(* Logix 5000 project; controller BWFG_Project vendor 1 type 14 code 92 rev 20.13; software revision 20.04 *)

TASK MainTask (continuous, watchdog 500 ms) : MainProgram

MODULES
   Local : vendor 1 type 14 code 92 (ICP 5, rev 20.13)
      DNET_Scanner : vendor 1 type 12 code 14 (ICP 11, rev 7.3, Output RPI 20 ms, Input RPI 20 ms)
      Servo_Module : 1756-M02AE (ICP 12, rev 20.2, MotionAsync RPI 25 ms, MotionEvent RPI 1000 ms, MotionSync RPI 2 ms)
      Ethenet_Module : 1756-EN2T (Ethernet 10.100.88.20, ICP 9, rev 10.7)   // CLX Etherent Module
         PF70 : vendor 1 type 123 code 48 (Ethernet 10.100.88.53, rev 2.9, Output RPI 20 ms)
              PF70:O.DRIVELOGICRSLT_START   // ENET Speed Start
              PF70:O.DRIVELOGICRSLT_REVERSE   // ENET Rev Start
              PF70:O.DRIVELOGICRSLT_FORWARD   // Enet FWD Start
             : vendor 1 type 123 code 8192 (DPI 5, rev 5.2)
      DHRIO : 1756-DHRIO (ICP 10, rev 5.4, Input RPI 25 ms)
         Flex_Rack : 1794-ASB (RIO 0, rev 1.1, Output RPI 16 ms)   // Flex RIO Rack in Workcell
         Robot_Rack : 1794-ASB (RIO 8, rev 1.1, Output RPI 48 ms)
END_MODULES

VAR_GLOBAL   (* controller tags *)
   Amber_Stack_LT : ALIAS FOR Flex_Rack:O.Data[3].1;   // The Amber stack Light
   Auto_mode : BOOL;   // Auto Mode Trigger ON/OFF
   Axis_0 : AXIS_SERVO;
   B3 : DINT;   // Hold value for robot Info
        .4   // Lift Locate Lower Cycle (AUTO)
        .0   // Permit Auto Mode
        .3   // Pallet Discarge Cycle
        .5   // Lift locate lower cycle auto
   Barcode_char : SINT[12] := ([0] := 110, [1] := 114, [2] := 32, [3] := 32, [4] := 32, [5] := 32, [6] := 32, [7] := 32, [8] := 32, [9] := 32, [10] := 32, [11] := 32);   // Barcode scanned info
   Barcode_Delay : BOOL;   // Delay created for barcode to allow info to be scanned then sent
   Barcode_Display : SINT[12] := ([0] := 62, [1] := 66, [2] := -16, [3] := -16, [4] := -16, [5] := -16, [6] := -16, [7] := -16, [8] := -16, [9] := -16, [10] := -16, [11] := -16);   // display the barcode value after info been translated from Asscii to decimal
   Barcode_OneShot : BOOL;   // a Oneshot for barcode to be sent
   Barcode_PB : BOOL;   // Push Button to Trigger the Barcode For manual mode and testing
   Barcode_Raw : STRING;   // Barcode Raw data (in ASCII)
   Barcode_Read_Done : BOOL := 1;   // Barcode signal it's done scanning
   Binary : DINT;
   Bottle_Control : CONTROL := (LEN := 5, EM := 1);   // Control for Bottle FiFo
   Bottle_FIFO : SINT[5];   // Bottle Fifo to Hold and send the list of Bottle value info (diffrent types of 12)
   BottleType : INT;   // Type of Bottle Given to be drawned
   Cabernet_Total : REAL := 100.0;
   Cell_Power_ON : ALIAS FOR Flex_Rack:I.Data[0].0;   // Workcell Power On Input
   Cell_Stop_PB : ALIAS FOR Flex_Rack:I.Data[1].11;   // Workcell Stop PB
   Champagne_Total : REAL := 100.0;
   Clear_Out_Oneshot : BOOL;   // Clear the Outputs when switching manual entry modes
   Cycle_Complete : ALIAS FOR Robot_Rack:I.Data[0].2;   // Cycle Complete Signal
   Cycle_Start : ALIAS FOR Robot_Rack:O.Data[0].0;   // Cycle start Trigger
   Direction_Mask_Value : DINT := 47;   // the Diresctional Mask for the VFD to change it From Ethernet to Deffalt
   Display_N : DINT[12];
   Display_PV : DINT;   // the Display PV screen, used to change the screen
   DNET_MODE_Select : BOOL;
   Drive_Actual_FWD_Speed : REAL;   // Real Speed of the FWD of the driver (in HZ)
   Drive_Actual_REV_Speed : REAL;   // Real Speed of the REV of the driver (in HZ)
   Drive_REQ_SPD_A : REAL;   // Driver running Indicator
   Drive_Running_IND : BOOL;   // the speed request for the driver in HZ
   Drive_SPD_Request : REAL;
   ENET_FWD_Speed : DINT;   // the set fwd speed
   ENET_REV_Speed : DINT;   // The set REV speed
   Enet_speed_convert : DINT;
   Enet_Speed_HOLD : DINT;
   Ent_Stop_Bit : ALIAS FOR Flex_Rack:O.Data[3].5;   // Ethernet Stop BIT
   Entrance_Convr_Message : SINT := 1;   // PV1000+ Entrance Conveyor Message 1=Stopped, 2=Forward 3=Reverse
   Entrance_FWD_PB : BOOL;   // PV1000+ ENTRANCED CONVEYOR FORWARD PB MANUAL SCREEN
   Entrance_REV_PB : BOOL;   // PV1000+ ENTRANCED CONVEYOR REVERSE PB MANUAL SCREEN
   Entrance_Speed_FPM : REAL;   // PV1000+ ENTRANCE CONVEYOR SPEED FEET-PER-MIN
   Entrance_Speed_Select : SINT := 5;
        .0   // PV1000+ Entrance Conveyor VFD Speed Select Bit 0
        .1   // PV1000+ Entrance Conveyor VFD Speed Select Bit 1
        .2   // PV1000+ Entrance Conveyor VFD Speed Select Bit 2
   Entrance_Speed_Timer : TIMER := (PRE := 5000);   // 5 second timer (1/12 of a minute)
        .DN   // 5 second timer (1/12 of a minute)
   Entrance_Sprocket_Pulse_Prox : ALIAS FOR Flex_Rack:I.Data[0].13;   // ENTRANCE CONVEYOR SPROCKET PULSE PROX 1 PULSE = 0.842 INCHES
   Event_Driven_Timer : TIMER[14] := ([0].PRE := 500, [1].PRE := 500, [2].PRE := 1700, [3].PRE := 500, [4].PRE := 500, [5].PRE := 500, [6].PRE := 500, [7].PRE := 500, [8].PRE := 500, [9].PRE := 500, [10].PRE := 500, [11].PRE := 500, [12].PRE := 500, [13].PRE := 2000);
   fault_servo_Reset : BOOL;
   FIFO_Bottle_Input : SINT := -16;
   FIFO_Bottle_Output : SINT := 1;
   FIFO_Level_Input : SINT := 96;
   FIFO_Level_Output : SINT := 55;
   FIFO_Location_Input : SINT := 66;
   FIFO_Location_Output : SINT := 1;
   FIFO_Wine_Input : SINT := -16;
   FIFO_Wine_Output : SINT := 1;
   Fill_Hold_percent : REAL := -160.0;   // holds percent values to then be sent as a whole value
   Fill_Level : INT;
   Fully_stop : BOOL;   // E_Stop LT
   FWD_REV_Mode : BOOL := 1;   // 0=FWD 1= REV
   Gate_Convr_FWD_PB : BOOL;   // PV1000+ GATE CONVEYOR FORWARD PB MANUAL SCREEN
   Gate_Convr_Message : SINT := 1;   // PV1000+ Gate Conveyor Message Display 1=Stopped 2=Forward 3=Reverse
   Gate_Convr_REV_PB : BOOL;   // PV1000+ GATE CONVEYOR REVERSE PB MANUAL SCREEN
   Gate_FS : BOOL;
   Gate_FWD_Starter : ALIAS FOR Flex_Rack:O.Data[4].2;   // Gate Conveyor Forward Motor Starter
   Gate_FWD_Starter_Contact : ALIAS FOR Flex_Rack:I.Data[1].5;   // Gate Conveyor Auxilary Contact Motor Forward Starter
   Gate_PL : ALIAS FOR Flex_Rack:O.Data[4].4;
   Gate_REV_Starter : ALIAS FOR Flex_Rack:O.Data[4].3;   // Gate Conveyor Reverse Motor Starter
   Gate_REV_Starter_Contact : ALIAS FOR Flex_Rack:I.Data[1].6;   // Gate Conveyor Auxilary Contact Motor Reverse Starter
   Gate_RS : BOOL;
   GIN : ALIAS FOR Robot_Rack:O.Data[0];
   Go_to_Auto_PB : BOOL;   // PV1000+ AUTO SCREEN SELECTED
   GO_to_Display_PB : BOOL;   // PV1000+ DISPALY SCREEN SELECTED
   Go_to_Robot : BOOL;   // PV1000+ ROBOT SCREEN SELECTED
   Go_To_Speed : BOOL;
   Go_to_Tracking : BOOL;   // PV1000+ TRACKING SCREEN SELECTED
   Goto_Main_PB : BOOL;   // PV1000+ MAIN SCREEN SELECTED
   Goto_Manual_PB : BOOL;   // PV1000+ MANUAL SCREEN SELECTED
   Green_Stack_LT : ALIAS FOR Flex_Rack:O.Data[3].2;
   HMI_indexer : SINT;
   Home_PB : BOOL;
   In_Cycle : ALIAS FOR Robot_Rack:I.Data[0].1;
   Input_clear_oneshot : BOOL;
   Level_Control : CONTROL := (LEN := 5, EM := 1);
   Level_FIFO : SINT[5];
   Level_Percent : REAL := 5.5;
   Lift_Locate_DOWN_Prox : ALIAS FOR Flex_Rack:I.Data[1].3;   // Lift Locate Down Prox
   Lift_Locate_Lower_Prox : ALIAS FOR Flex_Rack:I.Data[1].3;
   Lift_Locate_Message : SINT := 1;   // PV1000+ Lift-Locate-Unit Message Display 1=Lowered, 2=Raised
   Lift_Locate_PB : BOOL;   // PV1000+ Lift Locate PB (maintained)
   Lift_Locate_Prox : ALIAS FOR Flex_Rack:I.Data[1].1;
   Lift_Locate_Raised_Prox : ALIAS FOR Flex_Rack:I.Data[1].2;
   Lift_Locate_UP_Prox : ALIAS FOR Flex_Rack:I.Data[1].2;   // Lift Locate UP Prox
   Lift_Lower_Solenoid : ALIAS FOR Flex_Rack:O.Data[4].1;   // Lift Locate Lower Solenoid
   Lift_Raise_Solenoid : ALIAS FOR Flex_Rack:O.Data[4].0;   // Lift Locate Raise Solenoid
   Load_PB : BOOL;
   Location : INT;
   Location_Control : CONTROL := (LEN := 5, EM := 1);
   Location_FIFO : SINT[5];
   LTU_B : BOOL;
   LTU_DOWN_Prox : ALIAS FOR Flex_Rack:I.Data[0].10;   // Lift-transfer-Unit Down Prox
   LTU_Lower_Prox : ALIAS FOR Flex_Rack:I.Data[0].10;
   LTU_Lower_Solenoid : ALIAS FOR Flex_Rack:O.Data[3].12;   // Lift-Transfer-Unit Lower Solenoid
   LTU_Message : SINT := 2;   // PV1000+ Lift-Transfer-Unit Message Display 1=Lowered, 2=Centre 3=Raised
   LTU_Mid : BOOL;
   LTU_Posn_Select : SINT := 2;
        .0   // PV1000+ LTU Position Selector Bit 0
        .1   // PV1000+ LTU Position Selector Bit 1
   LTU_Prox : ALIAS FOR Flex_Rack:I.Data[0].9;
   LTU_Raise_Solenoid : ALIAS FOR Flex_Rack:O.Data[3].11;   // Lift-Transfer-Unit Raise Solenoid
   LTU_Raised_Prox : ALIAS FOR Flex_Rack:I.Data[0].11;
   LTU_Top : BOOL;
   LTU_UP_Prox : ALIAS FOR Flex_Rack:I.Data[0].11;   // Lift-transfer-Unit UP Prox
   Main_Screen_Button : BOOL;   // PV1000+ MAIN SCREEN SELECTED
   Man_Barcode_ON : BOOL;   // Allows the barcode to be turn on when running in manual mode for testing
   Man_Bottle : DINT := 1;
   Man_Level : DINT := 55;
   Man_Load_PB : BOOL;   // Loads the manual enetry values
   Man_Location : DINT := 1;
   Man_Mode : BOOL;
   Man_Mode_ON : BOOL;   // PV1000+ MANUAL MODE INDICATOR
   Man_Wine : DINT := 1;
   Manual_Enty : BOOL := 1;   // allows manual entry for orders
   manual_Screen_button : BOOL;   // PV1000+ Manual SCREEN SELECTED
   Merlot_Total : REAL := 94.5;
   Motion_Group_One : MOTION_GROUP;
   MSG_Display_Num : COUNTER := (PRE := 300, ACC := 154);
   MSG_Timer : TIMER := (PRE := 50, ACC := 41, EN := 1, TT := 1);
   MSG_Timer_2 : TIMER := (PRE := 50, EN := 1, TT := 1);
   New_Message_Sent_N : ALIAS FOR Local:11:I.Data[0].15;
   One_Shot : BOOL;
   One_Shot_Mid : BOOL;
   One_Shot_Rise : BOOL;
   OneShot_Clear_bits : BOOL;
   pallet_at_gate : ALIAS FOR Flex_Rack:I.Data[2].4;
   PF70_Fault_Reset : BOOL;
   PF70_Feedback_Speed_FWD_Hz : REAL;
   PF70_Feedback_Speed_REV_Hz : REAL;
   PF70_Parameter_Value : INT[300] := ([2] := 400, [10] := 2358, [12] := 8337, [13] := 8339, [16] := -6, [17] := 57, [26] := 37, [27] := 6000, [28] := 9, [29] := 2009, [41] := 5750, [42] := 5, [43] := 600, [44] := 1700, [45] := 21, [46] := 1, [47] := 300, [48] := 356, [54] := 5750, [55] := 1300, [56] := 3, [61] := 3, [62] := 237, [63] := 25, [69] := 219, [70] := 219, [71] := 1150, [72] := 150, [82] := 700, [83] := 100, [90] := 1, [91] := 700, [93] := 22, [94] := 700, [96] := 1, [97] := 600, [100] := 100, [101] := 50, [102] := 100, [103] := 200, [104] := 300, [105] := 400, [106] := 500, [107] := 600, [117] := 2, [119] := 600, [121] := 1000, [122] := 400, [127] := 5000, [128] := 4866, [129] := 200, [130] := 100, [131] := -1300, [132] := 1300, [140] := 5, [141] := 100, [142] := 5, [143] := 100, [148] := 14, [149] := 250,
        [150] := 3, [151] := 4, [155] := 1, [158] := 9, [160] := 450, [161] := 257, [162] := 260, [163] := 256, [170] := 4000, [175] := 10, [185] := 5, [192] := 1, [195] := 10, [196] := 1, [201] := 1, [202] := 2, [203] := -17715, [209] := 24204, [213] := 15, [214] := 273, [215] := 256, [216] := 40, [218] := 325, [226] := 8344, [227] := 24076, [234] := 499, [236] := 499, [238] := 74, [241] := 1, [242] := -17928, [243] := 75, [244] := -17383, [245] := 75, [246] := 28012, [247] := 75, [248] := 24586, [249] := 75, [250] := 22941, [259] := 959, [271] := 20497, [272] := 10082, [276] := 47, [277] := 47, [278] := 47, [279] := 47, [280] := 47, [281] := 47, [282] := 47, [283] := 47, [284] := 47, [285] := 15, [288] := 1, [291] := 1, [292] := 1);
   PF70_VFD_Control_Mode : SINT;   // VFD Control Mode 0=DIgital / 1 = ENET
   PO_BIT : BOOL;
   pos_add : DINT := 1;
   Postion_montior : INT;
   Postion_reset_Oneshot : BOOL := 1;
   Prestop_Lower_Solenoid : ALIAS FOR Flex_Rack:O.Data[3].10;   // PRESTOP LOWER SOLENOID COIL
   Prestop_Lower_Solenoid_MAN : BOOL;
   Prestop_Message : SINT := 2;   // PV1000+ Pre Stop Message Display 1=Down, 2=UP
   Prestop_PB : BOOL;   // PV1000+ PRE-STOP PB (maintained type) MANUAL SCREEN
   Prestop_Prox : ALIAS FOR Flex_Rack:I.Data[0].8;
   Product_Code : ALIAS FOR Robot_Rack:O.Data[1];
   Pushbutton_Index : BOOL;
   RAW_CELL_Number : INT;
   RED_Stack_LT : ALIAS FOR Flex_Rack:O.Data[3].0;
   Redi_Start_PB_N : ALIAS FOR Local:11:I.Data[15].1;
   Reset_FIFO : BOOL;
   Rest_Seq : BOOL;
   Return_Speed : ALIAS FOR PF70_Parameter_Value[2];   // speed refrence in frequancy
   Robot_Auto_Pass : BOOL := 1;   // allow sequance to work if robot is ready and clear or if bypass is on
   Robot_Bypass : BOOL;   // Skips Robot in sequance if ON
   Robot_Bypass_PB : BOOL;   // Robot Baypass button allowing robot to be skiped
   Robot_Clear : ALIAS FOR Robot_Rack:I.Data[0].0;   // checks if robot is clear of orignal program and is ready to start
   Robot_Cycle_Start : ALIAS FOR Robot_Rack:O.Data[0].0;
   Robot_Message : SINT;
   Robot_Product_Code : DINT;
   RPM : REAL := 200.0;
   Run_mode : ALIAS FOR Local:11:O.CommandRegister.Run;
   Screen_Number : DINT;   // SCREEN NUMBER FOR PV1000+ HMI
   Send_Next_Data_N : ALIAS FOR Local:11:O.Data[0].7;
   Seq_ON : BOOL;
   Seq_start : BOOL;
   Seq_Step : DINT[14] := ([1] := 278529, [2] := 278528, [3] := 278532, [4] := 278528, [5] := 8, [6] := 5576, [7] := 40, [8] := 72, [9] := 5064, [10] := 16, [11] := 16400, [13] := 22);
   Seq_Stop : BOOL;
   Sequencer_Output : DINT := 278529;
        .0   // Sequencer output bits 0
        .14   // Sequencer output bits 14
   Servo_ACC : INT := 25;
   Servo_Control : MOTION_INSTRUCTION[10] := ([0].FLAGS := 33554432, [1].FLAGS := -1610612736, [1].EN := 1, [1].DN := 1, [1].STATUS := 2, [1].STATE := 1, [2].FLAGS := 33554432, [3].FLAGS := 33554432, [4].FLAGS := 33554432);
        [2]   // Turn On Servo
        [1]   // Turn Off servo
        [0]   // Fault Resets Servo
        [3]   // Sends Servo Home
        [4]   // Sends Servo to Given Location based on Fill %
   Servo_Dec : INT := 25;
   Servo_Postion : REAL := 4.125;
   Servo_Speed : INT := 50;
   Servo_Sys_Fault : ALIAS FOR Axis_0.PhysicalAxisFault;
   Speed_Select_Conferm : BOOL;
   Sprocket_Pulse_Count : COUNTER := (PRE := 10000);   // COUNT SPROCKET PULSES IN TIME PERIOD
   SQO_Control : CONTROL := (LEN := 11, POS := 1, EN := 1);
   SQO_Mask : DINT := 287309823;
   Start_PB_PV1000 : BOOL;   // PV1000+ Start PB MANUAL SCREEN
   Status_Message : ALIAS FOR Robot_Rack:I.Data[1];
   Stop_PB_PV1000 : BOOL := 1;   // PV1000+ Stop PB MANUAL SCREEN
   System_On : BOOL;
   test_PB : BOOL := 1;
   Tigger_Barcode_N : ALIAS FOR Local:11:O.Data[0].0;
   timer_barcode : TIMER := (PRE := 50);
   Timer_Flash : TIMER[4] := ([0].PRE := 1000, [1].PRE := 1000, [2].PRE := 1000);
   Timer_Index_timer : TIMER := (PRE := 1000);
   Timer_Preset : DINT[31] := ([0] := 1000, [1] := 1000, [2] := 8000, [3] := 2000, [4] := 4000, [5] := 1000, [6] := 6500, [7] := 1000, [8] := 1000, [9] := 8000, [10] := 1000, [11] := 4000, [12] := 1000, [13] := 12000);
   timer_stop : DINT;
   Trains_FS : BOOL;
   Trains_RS : BOOL;
   Trans_Convr_FWD : ALIAS FOR Flex_Rack:O.Data[3].14;   // TRANSFER CONVEYOR FORWARD STARTER COIL
   Trans_Convr_FWD_MAN : BOOL;
   Trans_Convr_FWD_PB : BOOL;   // PV1000+ TRANSFER CONVEYOR FORWARD PB MANUAL SCREEN
   Trans_Convr_Message_PV1000 : DINT := 1;   // PV1000+ TRANSFER CONVEYOR MESSAGE DISPLAY 1=Stopped, 2=Forward 3=Reverse
   Trans_Convr_REV : ALIAS FOR Flex_Rack:O.Data[3].15;   // TRANSFER CONVEYOR REVERSE STARTER COIL
   Trans_Convr_REV_MAN : BOOL;
   Trans_Convr_REV_PB : BOOL;   // PV1000+ TRANSFER CONVEYOR REVERSE PB MANUAL SCREEN
   Trans_FWD_Starter_Contact : ALIAS FOR Flex_Rack:I.Data[0].14;   // Transfer Conveyor Auxilary Contact Motor Forward Starter
   Trans_REV_Starter_Contact : ALIAS FOR Flex_Rack:I.Data[0].15;   // Transfer Conveyor Auxilary Contact Motor Reverse Starter
   Transfer_Prestop_Prox : ALIAS FOR Flex_Rack:I.Data[1].8;
   Unload_PB : BOOL;
   Variables : SINT[12];
   VFD_FWD_Hold : SINT := 5;
   VFD_Message : MESSAGE;
        MessageParameters(ServiceCode := 16#000e, DestinationTag := PF70_Parameter_Value, ...)
   VFD_Message_2 : MESSAGE;
        MessageParameters(ServiceCode := 16#0010, LocalElement := Direction_Mask_Value, ...)
   VFD_REV_Bit : ALIAS FOR Flex_Rack:O.Data[3].6;   // ENTRANCED CONVEYOR VFD REVERSE BIT
   VFD_REV_Hold : SINT := 5;
   VFD_REV_MAN : BOOL;
   VFD_Speed_Bit_1 : ALIAS FOR Flex_Rack:O.Data[3].7;   // ENTRANCE CONVEYOR VFD SPEED 1 BIT
   VFD_Speed_Bit_2 : ALIAS FOR Flex_Rack:O.Data[3].8;   // ENTRANCE CONVEYOR VFD SPEED 1 BIT
   VFD_Speed_Bit_3 : ALIAS FOR Flex_Rack:O.Data[3].9;   // ENTRANCE CONVEYOR VFD SPEED 1 BIT
   VFD_Start_Bit : ALIAS FOR Flex_Rack:O.Data[3].4;   // ENTRANCE CONVEYOR VFD START BIT
   VFD_Start_MAN : BOOL;
   VFD_Stop_Bit : ALIAS FOR Flex_Rack:O.Data[3].5;   // ENTRANCED CONVEYOR VFD STOP BIT
   VFD_Stop_MAN : BOOL;
   VFD_Timer : TIMER := (PRE := 250);   // ENTRANCE VFD START BIT DELAY
   Wine_Control : CONTROL := (LEN := 5, EM := 1);
   Wine_FIFO : SINT[5];
   Wine_One_Shot : BOOL := 1;
   Wine_Total_1 : BOOL;
   Wine_Total_2 : BOOL;
   Wine_Total_3 : BOOL;
   Winetype : INT;
   Work_Cell_Number : SINT;
END_VAR

PROGRAM MainProgram   (* main routine MainRoutine *)
VAR
   DIV_01 : FBD_MATH := (SourceB := 17644.0);
   DIV_02 : FBD_MATH := (SourceB := 17644.0);
   MUL_01 : FBD_MATH := (SourceB := 252.05714);
   MUL_02 : FBD_MATH := (SourceB := 70.0);
   MUL_03 : FBD_MATH := (SourceB := 70.0);
   MVMT_01 : FBD_MASKED_MOVE;
   Sequencer : DINT;
END_VAR

ROUTINE Barcode   (* ladder *)
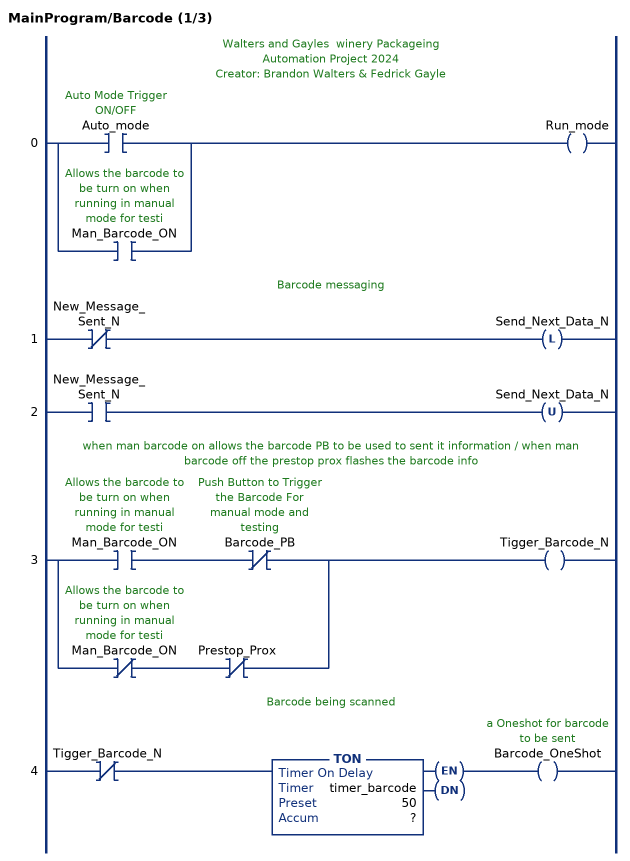
   // Walters and Gayles  winery Packageing
   // Automation Project 2024
   // Creator: Brandon Walters & Fedrick Gayle
   0: [XIC(Auto_mode) ,XIC(Man_Barcode_ON) ]OTE(Run_mode);
   // Barcode messaging
   1: XIO(New_Message_Sent_N)OTL(Send_Next_Data_N);
   2: XIC(New_Message_Sent_N)OTU(Send_Next_Data_N);
   // when man barcode on allows the barcode PB to be used to sent it information / when man barcode off the prestop prox flashes the barcode info
   3: [XIC(Man_Barcode_ON) XIO(Barcode_PB) ,XIO(Man_Barcode_ON) XIO(Prestop_Prox) ]OTE(Tigger_Barcode_N);
   // Barcode being scanned
   4: XIO(Tigger_Barcode_N)TON(timer_barcode,?,?)OTE(Barcode_OneShot);
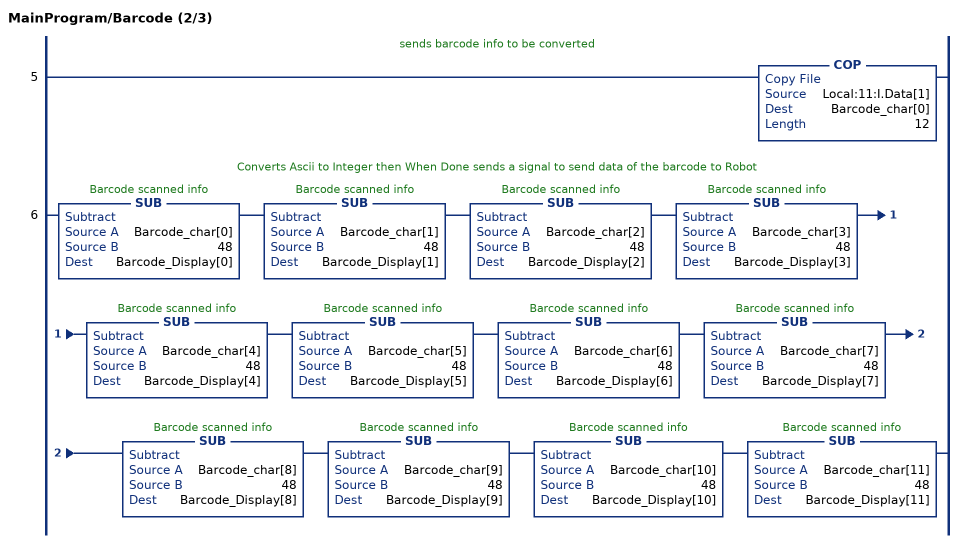
   // sends barcode info to be converted
   5: COP(Local:11:I.Data[1],Barcode_char[0],12);
   // Converts Ascii to Integer then When Done sends a signal to send data of the barcode to Robot
   6: SUB(Barcode_char[0],48,Barcode_Display[0])SUB(Barcode_char[1],48,Barcode_Display[1])SUB(Barcode_char[2],48,Barcode_Display[2])SUB(Barcode_char[3],48,Barcode_Display[3])SUB(Barcode_char[4],48,Barcode_Display[4])SUB(Barcode_char[5],48,Barcode_Display[5])SUB(Barcode_char[6],48,Barcode_Display[6])SUB(Barcode_char[7],48,Barcode_Display[7])SUB(Barcode_char[8],48,Barcode_Display[8])SUB(Barcode_char[9],48,Barcode_Display[9])SUB(Barcode_char[10],48,Barcode_Display[10])SUB(Barcode_char[11],48,Barcode_Display[11]);
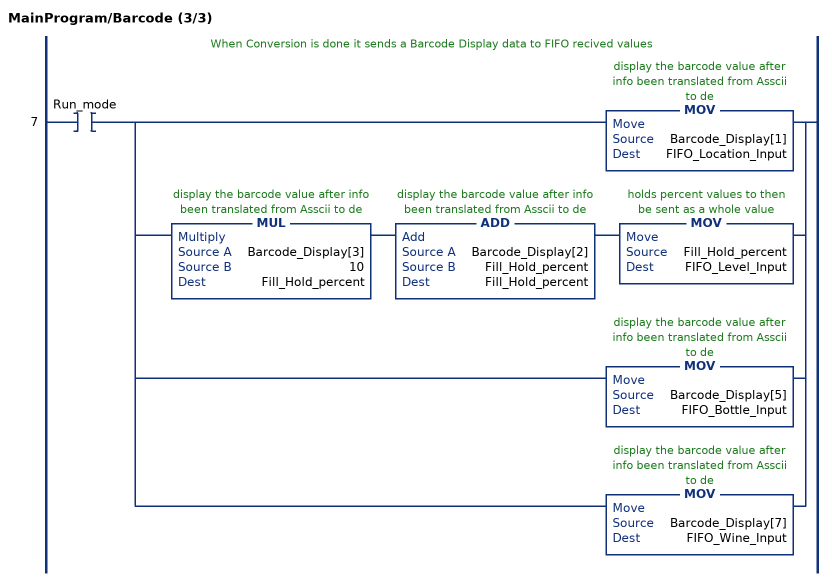
   // When Conversion is done it sends a Barcode Display data to FIFO recived values
   7: XIC(Run_mode)[MOV(Barcode_Display[1],FIFO_Location_Input) ,MUL(Barcode_Display[3],10,Fill_Hold_percent) ADD(Barcode_Display[2],Fill_Hold_percent,Fill_Hold_percent) MOV(Fill_Hold_percent,FIFO_Level_Input) ,MOV(Barcode_Display[5],FIFO_Bottle_Input) ,MOV(Barcode_Display[7],FIFO_Wine_Input) ];
END_ROUTINE

ROUTINE FIFO   (* ladder *)
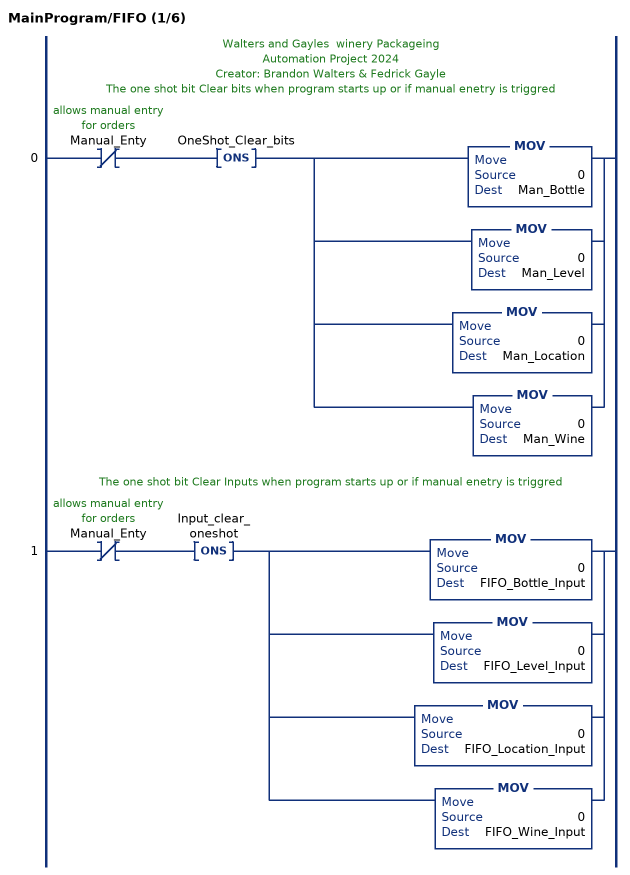
   // Walters and Gayles  winery Packageing
   // Automation Project 2024
   // Creator: Brandon Walters & Fedrick Gayle
   // The one shot bit Clear bits when program starts up or if manual enetry is triggred
   0: XIO(Manual_Enty)ONS(OneShot_Clear_bits)[MOV(0,Man_Bottle) ,MOV(0,Man_Level) ,MOV(0,Man_Location) ,MOV(0,Man_Wine) ];
   // The one shot bit Clear Inputs when program starts up or if manual enetry is triggred
   1: XIO(Manual_Enty)ONS(Input_clear_oneshot)[MOV(0,FIFO_Bottle_Input) ,MOV(0,FIFO_Level_Input) ,MOV(0,FIFO_Location_Input) ,MOV(0,FIFO_Wine_Input) ];
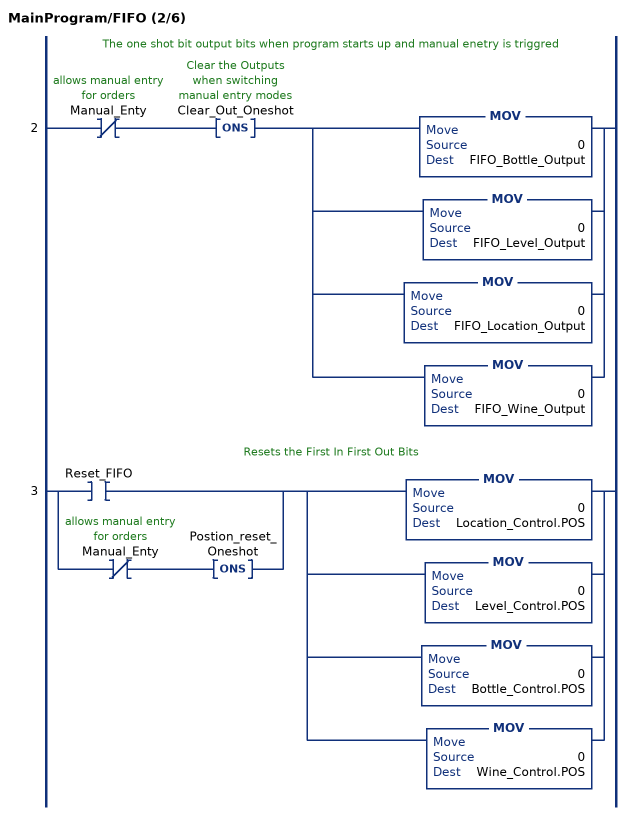
   // The one shot bit output bits when program starts up and manual enetry is triggred
   2: XIO(Manual_Enty)ONS(Clear_Out_Oneshot)[MOV(0,FIFO_Bottle_Output) ,MOV(0,FIFO_Level_Output) ,MOV(0,FIFO_Location_Output) ,MOV(0,FIFO_Wine_Output) ];
   // Resets the First In First Out Bits
   3: [XIC(Reset_FIFO) ,XIO(Manual_Enty) ONS(Postion_reset_Oneshot) ][MOV(0,Location_Control.POS) ,MOV(0,Level_Control.POS) ,MOV(0,Bottle_Control.POS) ,MOV(0,Wine_Control.POS) ];
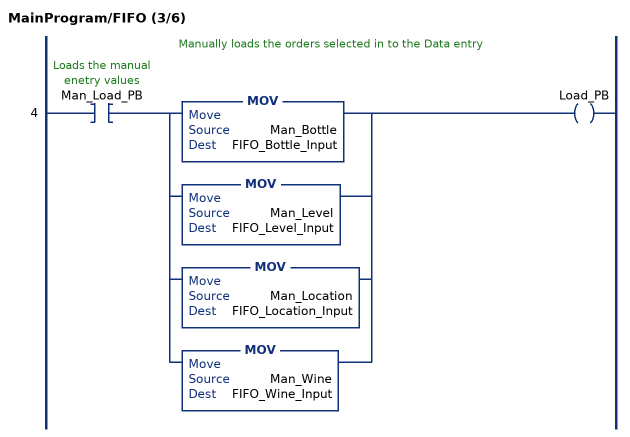
   // Manually loads the orders selected in to the Data entry
   4: XIC(Man_Load_PB)[MOV(Man_Bottle,FIFO_Bottle_Input) ,MOV(Man_Level,FIFO_Level_Input) ,MOV(Man_Location,FIFO_Location_Input) ,MOV(Man_Wine,FIFO_Wine_Input) ]OTE(Load_PB);
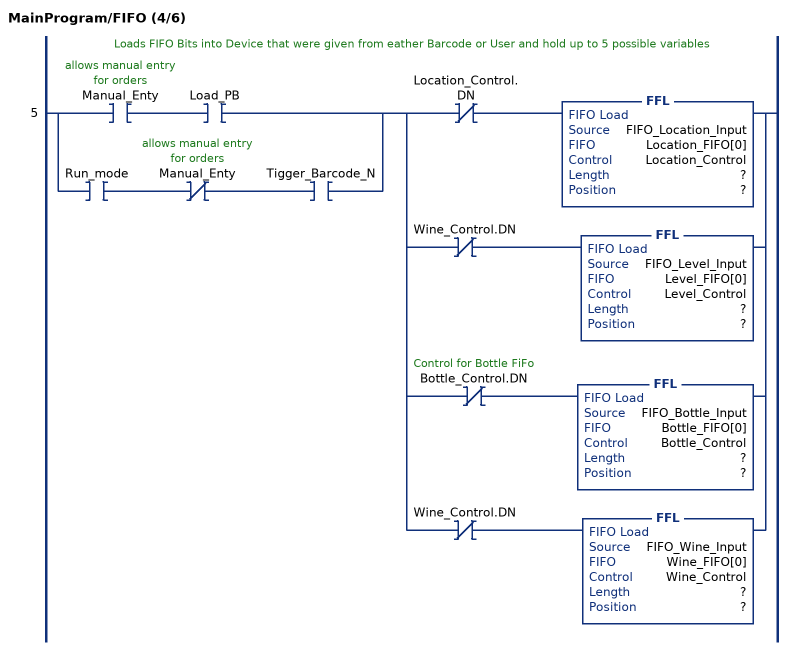
   // Loads FIFO Bits into Device that were given from eather Barcode or User and hold up to 5 possible variables
   5: [XIC(Manual_Enty) XIC(Load_PB) ,XIC(Run_mode) XIO(Manual_Enty) XIC(Tigger_Barcode_N) ][XIO(Location_Control.DN) FFL(FIFO_Location_Input,Location_FIFO[0],Location_Control,?,?) ,XIO(Wine_Control.DN) FFL(FIFO_Level_Input,Level_FIFO[0],Level_Control,?,?) ,XIO(Bottle_Control.DN) FFL(FIFO_Bottle_Input,Bottle_FIFO[0],Bottle_Control,?,?) ,XIO(Wine_Control.DN) FFL(FIFO_Wine_Input,Wine_FIFO[0],Wine_Control,?,?) ];
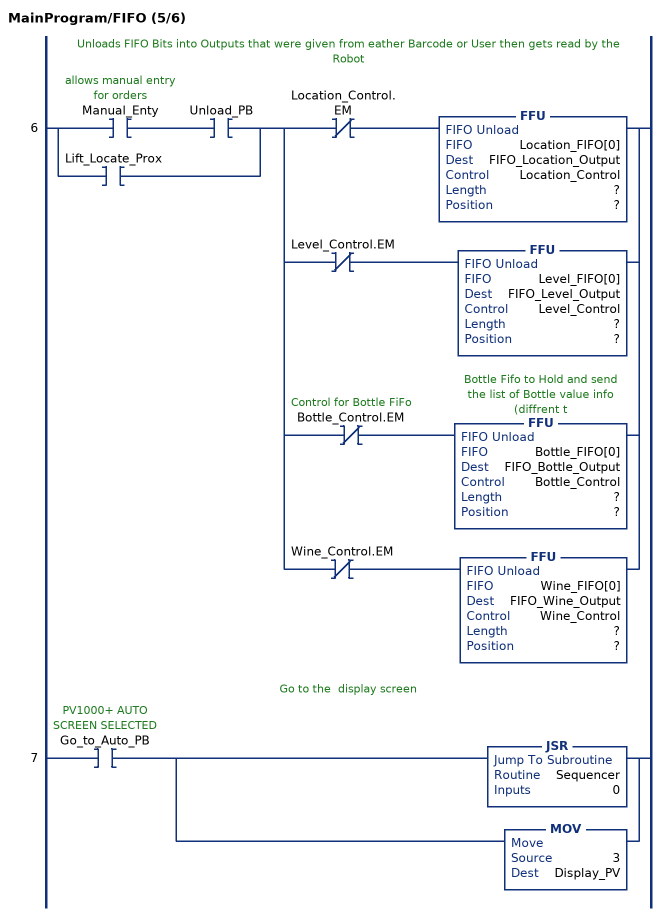
   // Unloads FIFO Bits into Outputs that were given from eather Barcode or User then gets read by the Robot
   6: [XIC(Manual_Enty) XIC(Unload_PB) ,XIC(Lift_Locate_Prox) ][XIO(Location_Control.EM) FFU(Location_FIFO[0],FIFO_Location_Output,Location_Control,?,?) ,XIO(Level_Control.EM) FFU(Level_FIFO[0],FIFO_Level_Output,Level_Control,?,?) ,XIO(Bottle_Control.EM) FFU(Bottle_FIFO[0],FIFO_Bottle_Output,Bottle_Control,?,?) ,XIO(Wine_Control.EM) FFU(Wine_FIFO[0],FIFO_Wine_Output,Wine_Control,?,?) ];
   // Go to the  display screen
   7: XIC(Go_to_Auto_PB)[JSR(Sequencer,0) ,MOV(3,Display_PV) ];
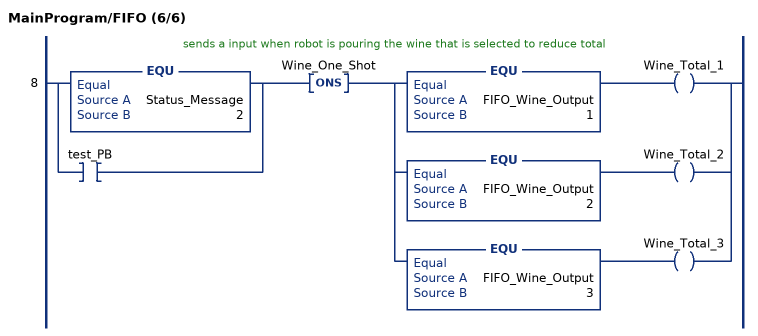
   // sends a input when robot is pouring the wine that is selected to reduce total
   8: [EQU(Status_Message,2) ,XIC(test_PB) ]ONS(Wine_One_Shot)[EQU(FIFO_Wine_Output,1) OTE(Wine_Total_1) ,EQU(FIFO_Wine_Output,2) OTE(Wine_Total_2) ,EQU(FIFO_Wine_Output,3) OTE(Wine_Total_3) ];
END_ROUTINE

ROUTINE HMI_Messages   (* ladder *)
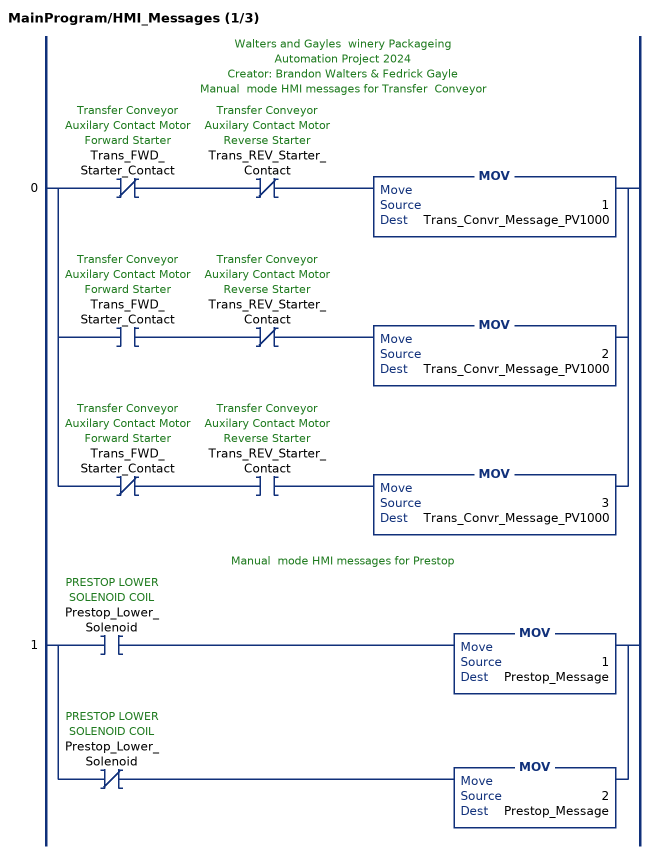
   // Walters and Gayles  winery Packageing
   // Automation Project 2024
   // Creator: Brandon Walters & Fedrick Gayle
   // Manual  mode HMI messages for Transfer  Conveyor
   0: [XIO(Trans_FWD_Starter_Contact) XIO(Trans_REV_Starter_Contact) MOV(1,Trans_Convr_Message_PV1000) ,XIC(Trans_FWD_Starter_Contact) XIO(Trans_REV_Starter_Contact) MOV(2,Trans_Convr_Message_PV1000) ,XIO(Trans_FWD_Starter_Contact) XIC(Trans_REV_Starter_Contact) MOV(3,Trans_Convr_Message_PV1000) ];
   // Manual  mode HMI messages for Prestop
   1: [XIC(Prestop_Lower_Solenoid) MOV(1,Prestop_Message) ,XIO(Prestop_Lower_Solenoid) MOV(2,Prestop_Message) ];
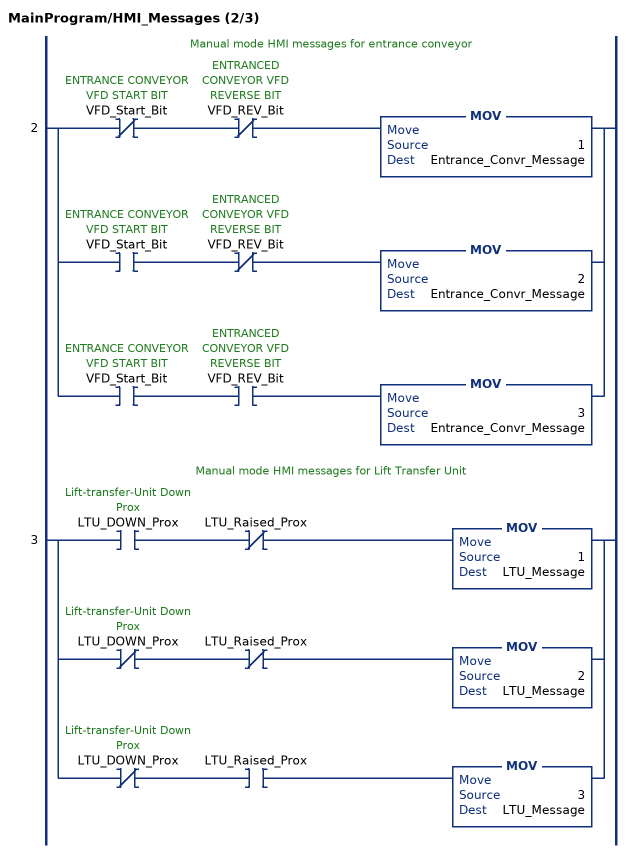
   // Manual mode HMI messages for entrance conveyor
   2: [XIO(VFD_Start_Bit) XIO(VFD_REV_Bit) MOV(1,Entrance_Convr_Message) ,XIC(VFD_Start_Bit) XIO(VFD_REV_Bit) MOV(2,Entrance_Convr_Message) ,XIC(VFD_Start_Bit) XIC(VFD_REV_Bit) MOV(3,Entrance_Convr_Message) ];
   // Manual mode HMI messages for Lift Transfer Unit
   3: [XIC(LTU_DOWN_Prox) XIO(LTU_Raised_Prox) MOV(1,LTU_Message) ,XIO(LTU_DOWN_Prox) XIO(LTU_Raised_Prox) MOV(2,LTU_Message) ,XIO(LTU_DOWN_Prox) XIC(LTU_Raised_Prox) MOV(3,LTU_Message) ];
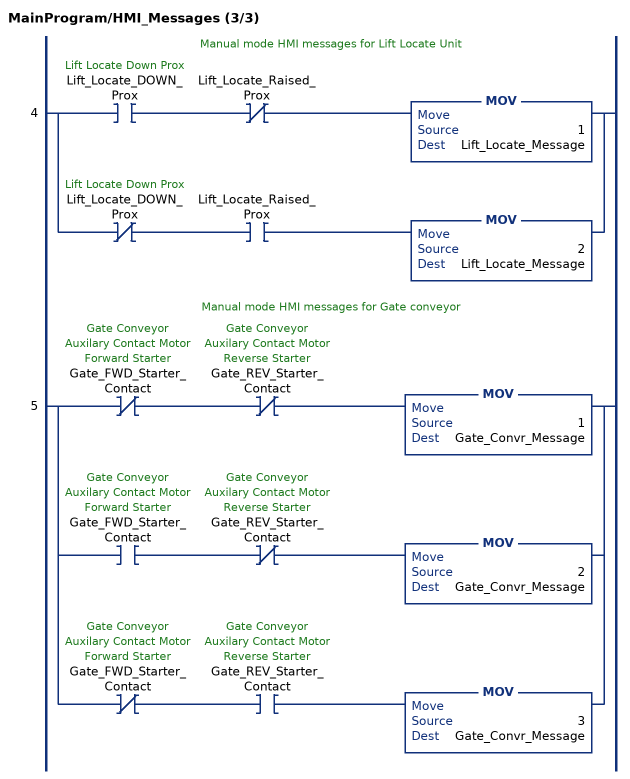
   // Manual mode HMI messages for Lift Locate Unit
   4: [XIC(Lift_Locate_DOWN_Prox) XIO(Lift_Locate_Raised_Prox) MOV(1,Lift_Locate_Message) ,XIO(Lift_Locate_DOWN_Prox) XIC(Lift_Locate_Raised_Prox) MOV(2,Lift_Locate_Message) ];
   // Manual mode HMI messages for Gate conveyor
   5: [XIO(Gate_FWD_Starter_Contact) XIO(Gate_REV_Starter_Contact) MOV(1,Gate_Convr_Message) ,XIC(Gate_FWD_Starter_Contact) XIO(Gate_REV_Starter_Contact) MOV(2,Gate_Convr_Message) ,XIO(Gate_FWD_Starter_Contact) XIC(Gate_REV_Starter_Contact) MOV(3,Gate_Convr_Message) ];
END_ROUTINE

ROUTINE MainRoutine   (* ladder *)
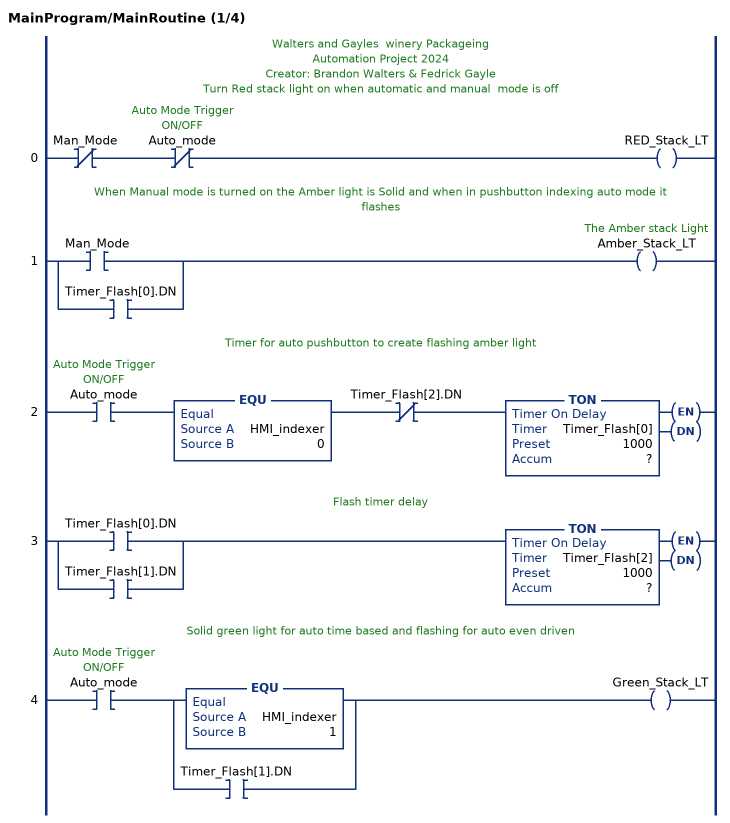
   // Walters and Gayles  winery Packageing
   // Automation Project 2024
   // Creator: Brandon Walters & Fedrick Gayle
   // Turn Red stack light on when automatic and manual  mode is off
   0: XIO(Man_Mode)XIO(Auto_mode)OTE(RED_Stack_LT);
   // When Manual mode is turned on the Amber light is Solid and when in pushbutton indexing auto mode it flashes
   1: [XIC(Man_Mode) ,XIC(Timer_Flash[0].DN) ]OTE(Amber_Stack_LT);
   // Timer for auto pushbutton to create flashing amber light
   2: XIC(Auto_mode)EQU(HMI_indexer,0)XIO(Timer_Flash[2].DN)TON(Timer_Flash[0],?,?);
   // Flash timer delay
   3: [XIC(Timer_Flash[0].DN) ,XIC(Timer_Flash[1].DN) ]TON(Timer_Flash[2],?,?);
   // Solid green light for auto time based and flashing for auto even driven
   4: XIC(Auto_mode)[EQU(HMI_indexer,1) ,XIC(Timer_Flash[1].DN) ]OTE(Green_Stack_LT);
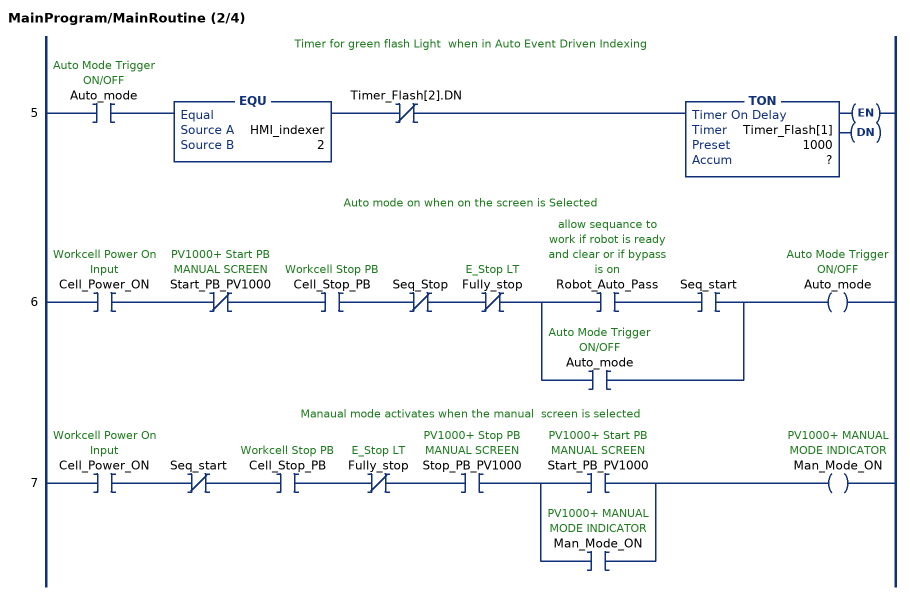
   // Timer for green flash Light  when in Auto Event Driven Indexing
   5: XIC(Auto_mode)EQU(HMI_indexer,2)XIO(Timer_Flash[2].DN)TON(Timer_Flash[1],?,?);
   // Auto mode on when on the screen is Selected
   6: XIC(Cell_Power_ON)XIO(Start_PB_PV1000)XIC(Cell_Stop_PB)XIO(Seq_Stop)XIO(Fully_stop)[XIC(Robot_Auto_Pass) XIC(Seq_start) ,XIC(Auto_mode) ]OTE(Auto_mode);
   // Manaual mode activates when the manual  screen is selected
   7: XIC(Cell_Power_ON)XIO(Seq_start)XIC(Cell_Stop_PB)XIO(Fully_stop)XIC(Stop_PB_PV1000)[XIC(Start_PB_PV1000) ,XIC(Man_Mode_ON) ]OTE(Man_Mode_ON);
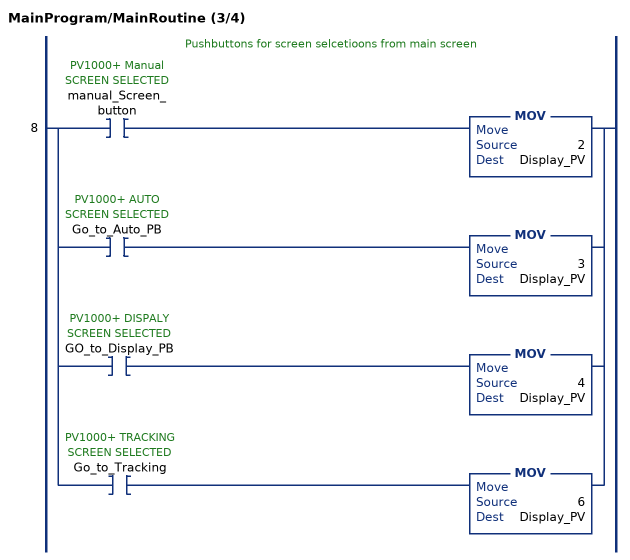
   // Pushbuttons for screen selcetioons from main screen
   8: [XIC(manual_Screen_button) MOV(2,Display_PV) ,XIC(Go_to_Auto_PB) MOV(3,Display_PV) ,XIC(GO_to_Display_PB) MOV(4,Display_PV) ,XIC(Go_to_Tracking) MOV(6,Display_PV) ];
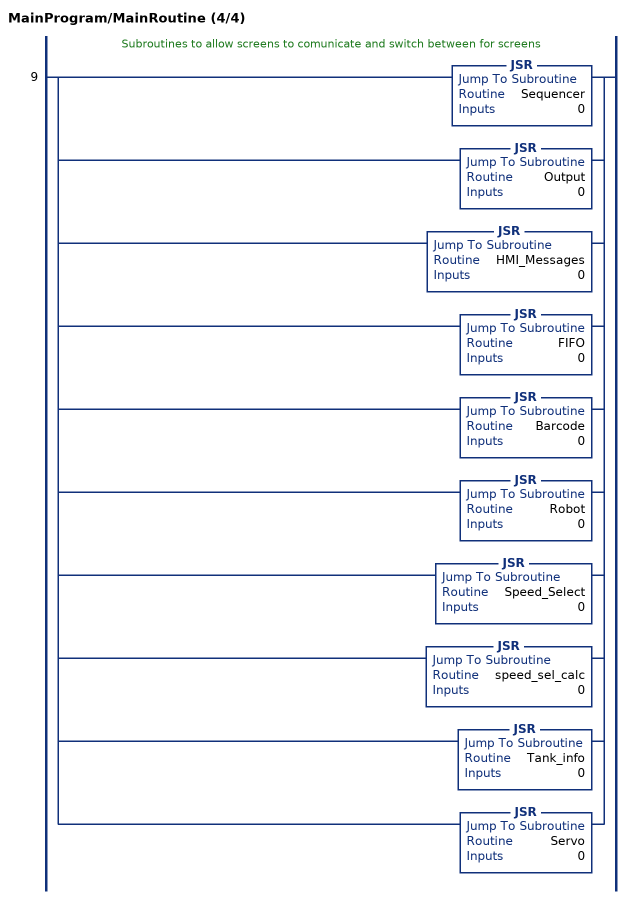
   // Subroutines to allow screens to comunicate and switch between for screens
   9: [JSR(Sequencer,0) ,JSR(Output,0) ,JSR(HMI_Messages,0) ,JSR(FIFO,0) ,JSR(Barcode,0) ,JSR(Robot,0) ,JSR(Speed_Select,0) ,JSR(speed_sel_calc,0) ,JSR(Tank_info,0) ,JSR(Servo,0) ];
END_ROUTINE

ROUTINE Output   (* ladder *)
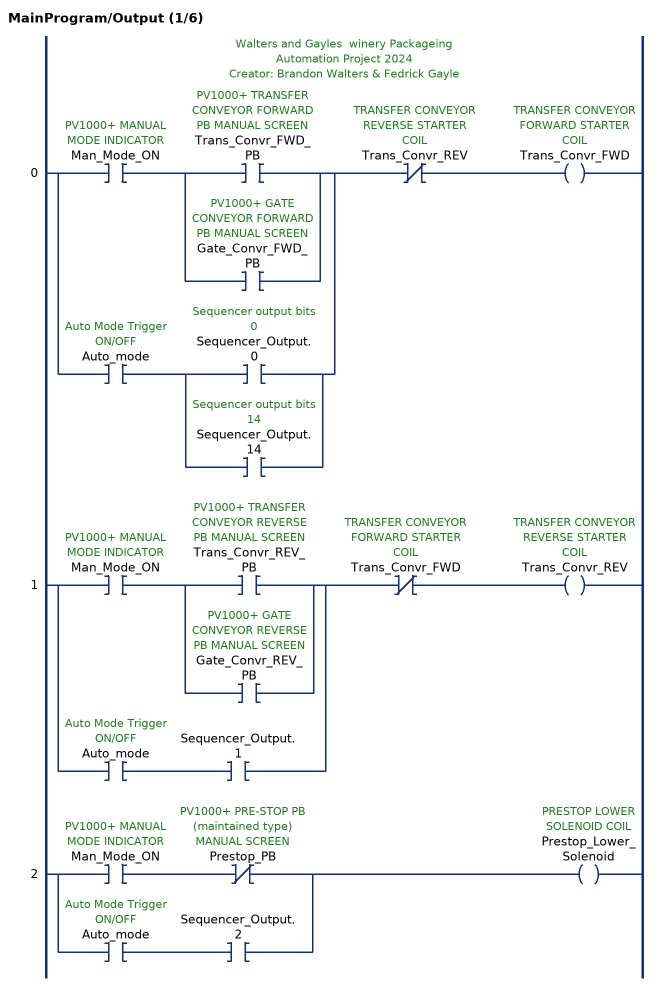
   // Walters and Gayles  winery Packageing
   // Automation Project 2024
   // Creator: Brandon Walters & Fedrick Gayle
   0: [XIC(Man_Mode_ON) [XIC(Trans_Convr_FWD_PB) ,XIC(Gate_Convr_FWD_PB) ] ,XIC(Auto_mode) [XIC(Sequencer_Output.0) ,XIC(Sequencer_Output.14) ] ]XIO(Trans_Convr_REV)OTE(Trans_Convr_FWD);
   1: [XIC(Man_Mode_ON) [XIC(Trans_Convr_REV_PB) ,XIC(Gate_Convr_REV_PB) ] ,XIC(Auto_mode) XIC(Sequencer_Output.1) ]XIO(Trans_Convr_FWD)OTE(Trans_Convr_REV);
   2: [XIC(Man_Mode_ON) XIO(Prestop_PB) ,XIC(Auto_mode) XIC(Sequencer_Output.2) ]OTE(Prestop_Lower_Solenoid);
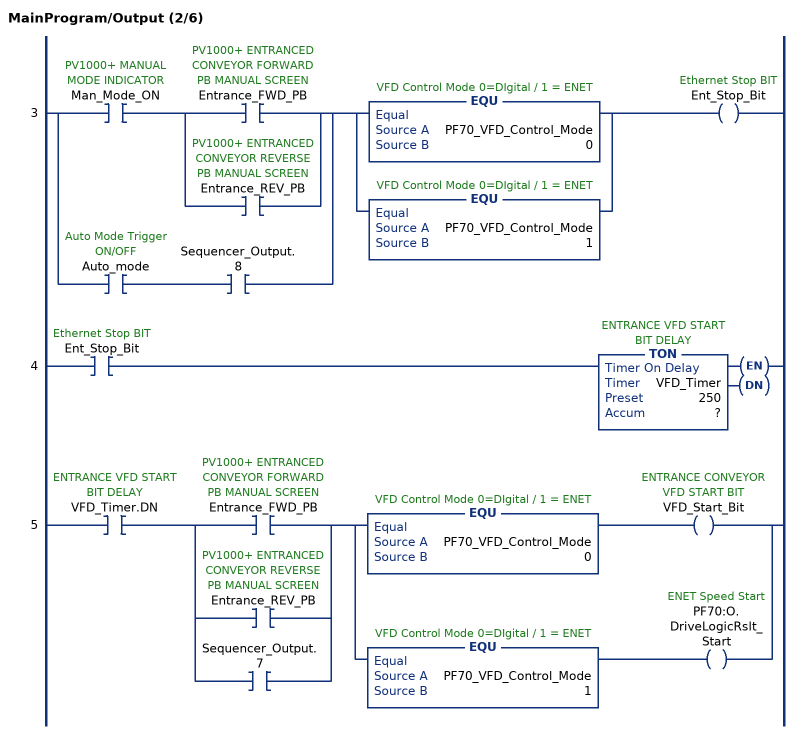
   3: [XIC(Man_Mode_ON) [XIC(Entrance_FWD_PB) ,XIC(Entrance_REV_PB) ] ,XIC(Auto_mode) XIC(Sequencer_Output.8) ][EQU(PF70_VFD_Control_Mode,0) ,EQU(PF70_VFD_Control_Mode,1) ]OTE(Ent_Stop_Bit);
   4: XIC(Ent_Stop_Bit)TON(VFD_Timer,?,?);
   5: XIC(VFD_Timer.DN)[XIC(Entrance_FWD_PB) ,XIC(Entrance_REV_PB) ,XIC(Sequencer_Output.7) ][EQU(PF70_VFD_Control_Mode,0) OTE(VFD_Start_Bit) ,EQU(PF70_VFD_Control_Mode,1) OTE(PF70:O.DriveLogicRslt_Start) ];
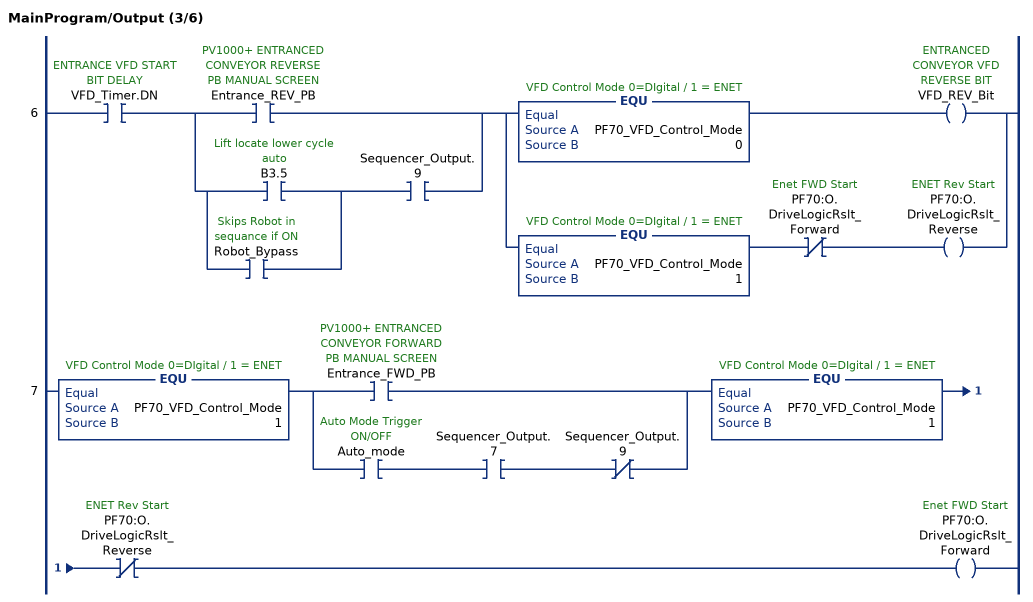
   6: XIC(VFD_Timer.DN)[XIC(Entrance_REV_PB) ,[XIC(B3.5) ,XIC(Robot_Bypass) ] XIC(Sequencer_Output.9) ][EQU(PF70_VFD_Control_Mode,0) OTE(VFD_REV_Bit) ,EQU(PF70_VFD_Control_Mode,1) XIO(PF70:O.DriveLogicRslt_Forward) OTE(PF70:O.DriveLogicRslt_Reverse) ];
   7: EQU(PF70_VFD_Control_Mode,1)[XIC(Entrance_FWD_PB) ,XIC(Auto_mode) XIC(Sequencer_Output.7) XIO(Sequencer_Output.9) ]EQU(PF70_VFD_Control_Mode,1)XIO(PF70:O.DriveLogicRslt_Reverse)OTE(PF70:O.DriveLogicRslt_Forward);
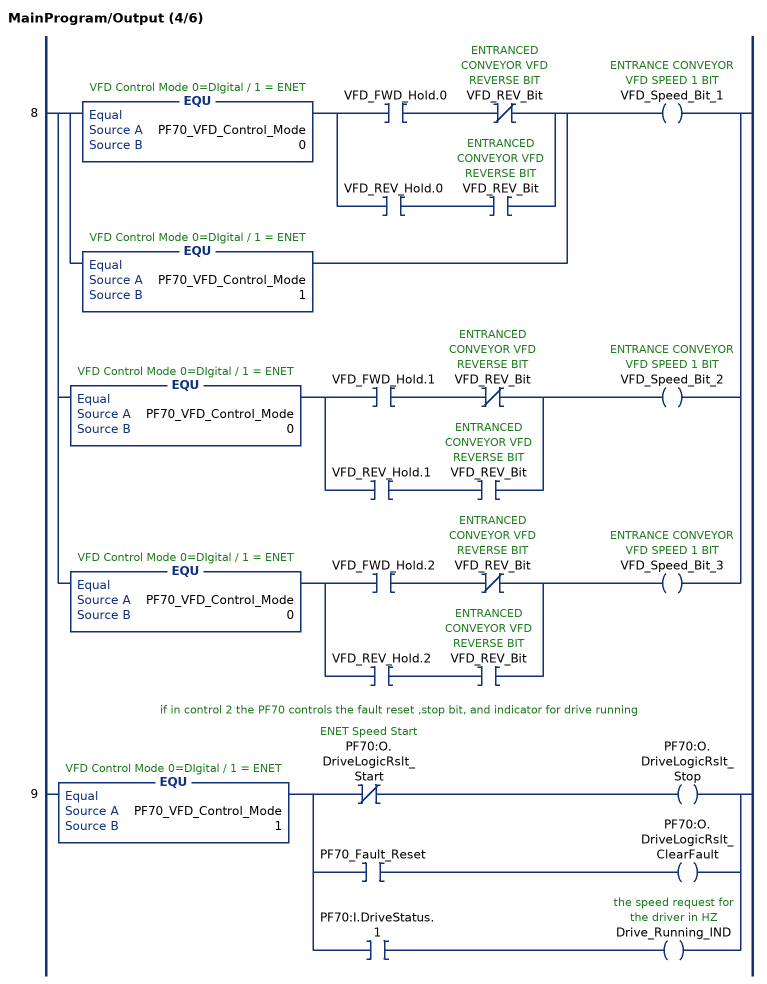
   8: [[EQU(PF70_VFD_Control_Mode,0) [XIC(VFD_FWD_Hold.0) XIO(VFD_REV_Bit) ,XIC(VFD_REV_Hold.0) XIC(VFD_REV_Bit) ] ,EQU(PF70_VFD_Control_Mode,1) ] OTE(VFD_Speed_Bit_1) ,EQU(PF70_VFD_Control_Mode,0) [XIC(VFD_FWD_Hold.1) XIO(VFD_REV_Bit) ,XIC(VFD_REV_Hold.1) XIC(VFD_REV_Bit) ] OTE(VFD_Speed_Bit_2) ,EQU(PF70_VFD_Control_Mode,0) [XIC(VFD_FWD_Hold.2) XIO(VFD_REV_Bit) ,XIC(VFD_REV_Hold.2) XIC(VFD_REV_Bit) ] OTE(VFD_Speed_Bit_3) ];
   // if in control 2 the PF70 controls the fault reset ,stop bit, and indicator for drive running
   9: EQU(PF70_VFD_Control_Mode,1)[XIO(PF70:O.DriveLogicRslt_Start) OTE(PF70:O.DriveLogicRslt_Stop) ,XIC(PF70_Fault_Reset) OTE(PF70:O.DriveLogicRslt_ClearFault) ,XIC(PF70:I.DriveStatus.1) OTE(Drive_Running_IND) ];
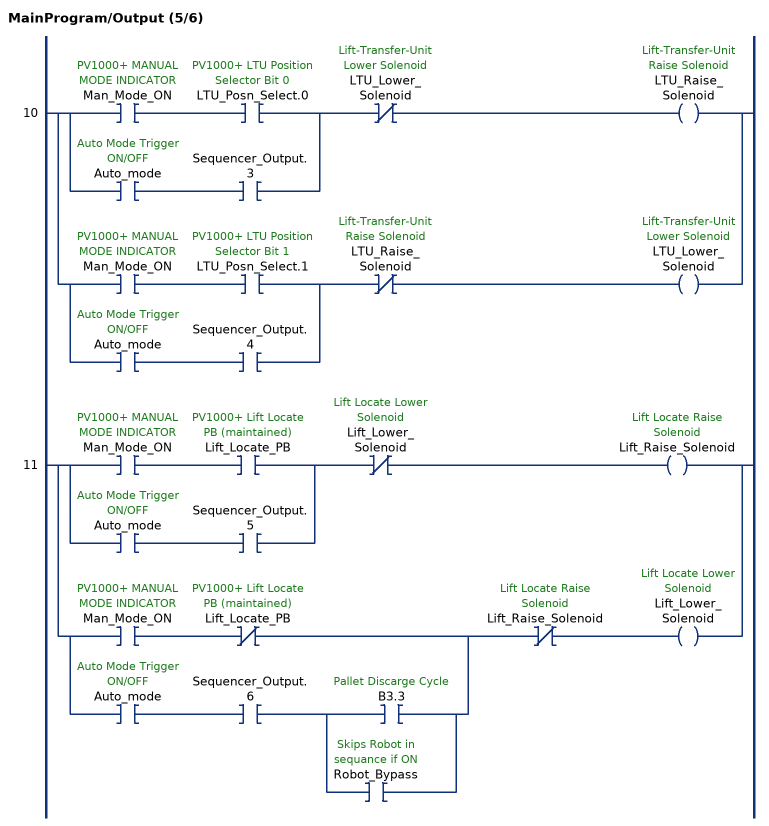
   10: [[XIC(Man_Mode_ON) XIC(LTU_Posn_Select.0) ,XIC(Auto_mode) XIC(Sequencer_Output.3) ] XIO(LTU_Lower_Solenoid) OTE(LTU_Raise_Solenoid) ,[XIC(Man_Mode_ON) XIC(LTU_Posn_Select.1) ,XIC(Auto_mode) XIC(Sequencer_Output.4) ] XIO(LTU_Raise_Solenoid) OTE(LTU_Lower_Solenoid) ];
   11: [[XIC(Man_Mode_ON) XIC(Lift_Locate_PB) ,XIC(Auto_mode) XIC(Sequencer_Output.5) ] XIO(Lift_Lower_Solenoid) OTE(Lift_Raise_Solenoid) ,[XIC(Man_Mode_ON) XIO(Lift_Locate_PB) ,XIC(Auto_mode) XIC(Sequencer_Output.6) [XIC(B3.3) ,XIC(Robot_Bypass) ] ] XIO(Lift_Raise_Solenoid) OTE(Lift_Lower_Solenoid) ];
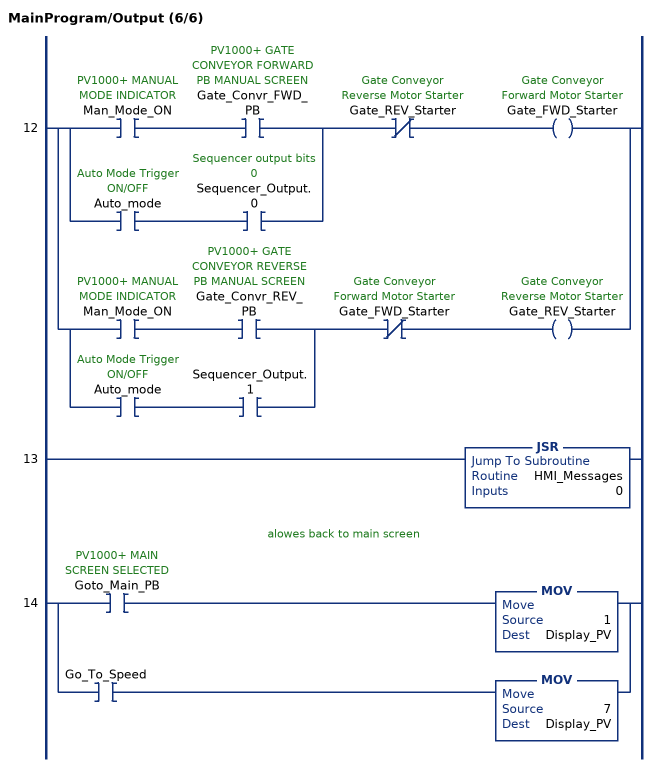
   12: [[XIC(Man_Mode_ON) XIC(Gate_Convr_FWD_PB) ,XIC(Auto_mode) XIC(Sequencer_Output.0) ] XIO(Gate_REV_Starter) OTE(Gate_FWD_Starter) ,[XIC(Man_Mode_ON) XIC(Gate_Convr_REV_PB) ,XIC(Auto_mode) XIC(Sequencer_Output.1) ] XIO(Gate_FWD_Starter) OTE(Gate_REV_Starter) ];
   13: JSR(HMI_Messages,0);
   // alowes back to main screen
   14: [XIC(Goto_Main_PB) MOV(1,Display_PV) ,XIC(Go_To_Speed) MOV(7,Display_PV) ];
END_ROUTINE
